TYPE T_CodeBATCH : STRING[10];
END_TYPE

(* stored: Version 1.1.0.1, ProductVersion 3.1.4024.15
   DUT T_CodeBATCH: Id {b3129944-4ddb-4b5f-9ef9-b6e719024768} *)
